Fanuc KAREL source: kd00073.KL

PROGRAM KD00073
%STACKSIZE=65535
%PRIORITY=65535
%NOLOCKGROUP
VAR
I : INTEGER
J : INTEGER
B : BOOLEAN
R : REAL
S : STRING[80]
BEGIN
I=0
I=(I + 1)
-- UNRESOLVED_PC line 13 opcodes [21 2E 5B 79] marker_code=36
END KD00073
